INTERFACE ITcoMomentaryTask EXTENDS ITcoObject

(*~
	<docu>
		<summary>
			Use to set the state of the '''TcoMomentaryOnTask''' to the value '''FALSE'''.
		</summary>			
	</docu>	
~*)
METHOD Off : BOOL
END_METHOD

(*~
	<docu>
		<summary>
			Use to set the state of the '''TcoMomentaryOnTask''' to the value '''TRUE'''.
		</summary>			
	</docu>	
~*)
METHOD On : BOOL
END_METHOD

END_INTERFACE

(* stored: Version 1.1.0.1
   Itf ITcoMomentaryTask: Id {5d9fd10b-53b1-0244-2e57-9b3a83ecb8b1}
   Method Off: Id {e72503c5-8318-0250-2de1-7cb22337cd30}
   Method On: Id {e3cd9904-f7e0-02ea-0c33-d78ab53b6239} *)
